VAR_GLOBAL CONSTANT
	nMAX_DATA_ELEMENTS : UINT := 100;
END_VAR

(* stored: Version 1.1.0.1, ProductVersion 3.1.4022.10
   GVL GVL_Constants: Id {c8178947-0536-41c7-b8c0-dc6291ef2c08} *)
